Staubli VAL3: page.pgx

public program page(string& x_sMenuName[], num x_nIndex)
// set all the page
begin
  // load the default one
  call language:page(x_sMenuName,x_nIndex)
end
